// TIA Portal V17 export
// export: Created 2025-06-26T07:49:15.8052087Z, ExportSetting WithDefaults, DisplayName Totally Integrated Automation Portal, DisplayVersion V17 Update 8, DisplayName TIA Portal Openness, DisplayVersion V17 Update 8, DisplayName TIA Portal Version Control Interface, DisplayVersion V17, DisplayName STEP 7 Professional, DisplayVersion V17 Update 8, DisplayName STEP 7 Safety, DisplayVersion V17 Update 6, DisplayName WinCC Advanced, DisplayVersion V17 Update 8
DATA_BLOCK "Puma_DB"   // DB4
VERSION : 0.1
// stored: AutoNumber true, DBAccessibleFromOPCUA true, InstanceOfName Puma, InstanceOfType FB
"Puma"
   // VAR_INPUT
   //    bEnable : Bool;
   // END_VAR
   // VAR
   //    Watchdog : "fbHeartbeatCount2";
   //    Dummy { S7_SetPoint := 'True'} : UInt;
   //    epForceExpansionValveSP : Bool;
   //    enForceExpansionValveSP : Bool;
   //    epForceHeatSinkOutSP : Bool;
   //    enForceHeatSinkOutSP : Bool;
   //    epForceMotorRpmSP : Bool;
   //    enForceMotorRpmSP : Bool;
   //    epForceOilHeatingSP : Bool;
   //    enForceOilHeatingSP : Bool;
   //    epForcePinchSP : Bool;
   //    enForcePinchSP : Bool;
   //    epForceSuperheatSP : Bool;
   //    enForceSuperheatSP : Bool;
   //    epStartRequest : Bool;
   //    enStartRequest : Bool;
   //    epStopRequest : Bool;
   //    enStopRequest : Bool;
   //    epAlarmAcknowledge : Bool;
   //    enAlarmAcknowledge : Bool;
   //    epResetEmergencyStop : Bool;
   //    enResetEmergencyStop : Bool;
   //    epHydrolockProtection : Bool;
   //    enHydrolockProtection : Bool;
   //    enClearance : Bool;
   //    ExpansionManualPrev : Real;
   //    HeatSinkManualPrev : Real;
   //    PerformanceManualPrev : Real;
   //    OilHeatingManualPrev : Real;
   //    PinchManualPrev : Real;
   //    SuperheatManualPrev : Real;
   //    WatchdogTimeout : TON_TIME;
   // END_VAR
BEGIN
END_DATA_BLOCK
